INTERFACE I_CyclicExecution

METHOD CyclicExecute : BOOL
VAR_INPUT
END_VAR
END_METHOD

END_INTERFACE

(* stored: Version 1.1.0.1, ProductVersion 3.1.4024.5
   Itf I_CyclicExecution: Id {2930f0cc-8ff3-40f0-a23a-2630be799c9e}
   Method CyclicExecute: Id {a6f77b5a-1b5c-4b6a-a4a6-f3e521dca4eb} *)
